RoboDK station: layout_PR2-2-7-bis.rdk

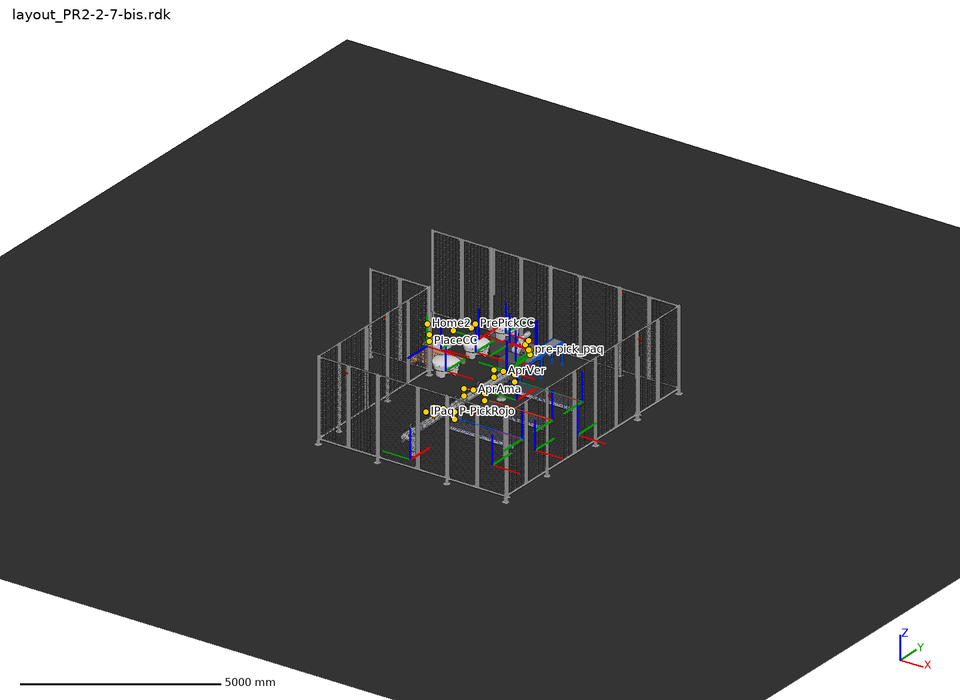
[picture v0: the station drawn from its stored meshes, robots at their saved joint values, targets as dots, program paths as lines]
Station def_pim_nigr (saved by RoboDK 5.9.4). Poses are relative to the parent item; angles as X-Y-Z fixed-axis rotations.
Station parameters (name, value as stored): IO_0, 1, IO_5, 1, IO_2, 1, IO_1, 1, IO_3, 0, 0, 0, 1, 0, 4, 0, SenyalSensor, 0, num_Pimiento, 0, num_Pimiento_Ama, 0, num_Pimiento_Rojo, 0, num_Pimiento_Verde, 0
  - folder Robots
    - frame D1Base at (200, 100, 1550) mm
      - robot D1 (model ABB IRB 360-1/1130 4D): 4 axes, payload 3 kg, reach 565 mm, repeatability 0.04 mm, weight 120 kg
          joint limits [-46.1, -46.1, -46.1, -36000] to [100.2, 100.2, 100.2, 36000]; home [0, 0, 0, 0]; saved at [70.365, 26.482, 30.889, 0]
        - tool GripR, TCP at (0, 0, 130) mm, size 75 x 83 x 136.1 mm
    - frame D2Base at (200, 1400, 1550) mm
      - robot D2 (model ABB IRB 360-1/1130 4D): 4 axes, payload 3 kg, reach 565 mm, repeatability 0.04 mm, weight 120 kg
          joint limits [-46.1, -46.1, -46.1, -36000] to [100.2, 100.2, 100.2, 36000]; home [0, 0, 0, 0]; saved at [70.365, 26.482, 30.889, 0]
        - tool GripA, TCP at (0, 0, 130) mm, size 75 x 83 x 136.1 mm
    - frame D3Base at (200, 2700, 1550) mm
      - robot D3 (model ABB IRB 360-1/1130 4D): 4 axes, payload 3 kg, reach 565 mm, repeatability 0.04 mm, weight 120 kg
          joint limits [-46.1, -46.1, -46.1, -36000] to [100.2, 100.2, 100.2, 36000]; home [0, 0, 0, 0]; saved at [70.365, 26.482, 30.889, 0]
        - tool GripV, TCP at (0, 0, 130) mm, size 75 x 83 x 136.1 mm
    - frame ABBPaq at (-570, 4240, -50) mm
      - robot ABBPaq (model ABB IRB 120-3/0.6): 6 axes, payload 3 kg, reach 580 mm, repeatability 0.01 mm, weight 25 kg
          modified DH rows (alpha deg, a mm, theta deg, d mm): 0, 0, 0, 290; -90, 0, -90, 0; 0, 270, 0, 0; -90, 70, 0, 302; 90, 0, 0, 0; -90, 0, 180, 72
          joint limits [-165, -110, -90, -160, -120, -400] to [165, 110, 70, 160, 120, 400]; home [0, 0, 0, 0, 0, 0]; saved at [84.8, 55.71, -70.13, 0, 104.39, 85]
        - tool ventosa_paq, TCP at (0, 0, 130) mm, size 75 x 83 x 136.1 mm
      - object Pedestal H24in (Type 1) at (-40, 0, -610) mm, size 400 x 400 x 609.6 mm, geometry from Pedestal-H24in-Type-1.sld
      - object SICK WL4S Laser Sensor at (638.65, -30.04, 245) mm, rotated rx 0 ry 0 rz 180 deg, size 683.3 x 45.2 x 12.5 mm, geometry from SICK-WL4S-Laser-Sensor.sld
    - frame ABBPallet at (-3120, 4660, -590) mm
      - robot ABBPallet (model ABB IRB 260): 4 axes, payload 30 kg, reach 1560 mm, repeatability 0.1 mm, weight 340 kg
          joint limits [-180, -28, -17, -300] to [180, 85, 119, 300]; home [0, 0, 0, 0]; saved at [-38.87, 11.87, -1.33, -35]
        - tool ventosa_pallet, TCP at (0, 30, 180) mm, size 239 x 147 x 184.9 mm
    - folder ProgCintas
      - program cintaROJO (3 instructions, listed below)
      - program cintaAMA (3 instructions, listed below)
      - program cintaVERDE (3 instructions, listed below)
  - folder Cintas
    - frame Conveyor Rojo at (2400, 300, 200) mm, rotated rx 0 ry 0 rz -180 deg
      - robot CRojo: 1 axes
          modified DH rows (alpha deg, a mm, theta deg, d mm): 0, 0, 0, 0 linear
          base shift (0, 0, 0) mm, rotated rx 0 ry 90 rz 0 deg
          joint limits [-500000] to [500000]; home [0]; saved at [0]
        - frame PRojo at (760, 220, -850) mm, rotated rx 0 ry 0 rz -180 deg
          - object PiRojo at (0, -5, 50) mm, rotated rx 180 ry 0 rz 180 deg, size 100 x 100 x 100 mm, geometry from Sphere-D100mm.sld
      - object SensorRojo at (1900, 0, 0) mm, rotated rx 0 ry 0 rz 90 deg, size 683.3 x 45.2 x 12.5 mm, geometry from SICK-WL4S-Laser-Sensor.sld
      - target IRojo (joint target) at (0, 0, 0) mm; joints [0] of CRojo
      - target FRojo (joint target) at (1900, 0, 0) mm; joints [1900] of CRojo
      - target P-PickRojo (Cartesian target) at (1900, 225, 300) mm, rotated rx 180 ry 0 rz 180 deg; joints [-31.271, 25.228, 30.105, 0] of D1
      - target PickRojo (Cartesian target) at (1900, 225, 100) mm, rotated rx 180 ry 0 rz 180 deg; joints [4.869, 47.636, 51.233, 0] of D1
      - target AprRojo (Cartesian target) at (2250, 225, 300) mm, rotated rx 180 ry 0 rz 180 deg; joints [4.316, -9.05, -2.968, 0] of D1
      - target P-PlaceRojo (Cartesian target) at (2532, 225, 250) mm, rotated rx 180 ry 0 rz 180 deg; joints [51.618, -4.676, 0.802, 0] of D1
      - target PlaceRojo (Cartesian target) at (2532, 225, 50) mm, rotated rx 180 ry 0 rz 180 deg; joints [70.365, 26.482, 30.889, 0] of D1
    - frame Conveyor Amarillo at (2400, 1600, 200) mm, rotated rx 0 ry 0 rz 180 deg
      - robot CAma: 1 axes
          modified DH rows (alpha deg, a mm, theta deg, d mm): 0, 0, 0, 0 linear
          base shift (0, 0, 0) mm, rotated rx 0 ry 90 rz 0 deg
          joint limits [-500000] to [500000]; home [0]; saved at [0]
        - frame PAma at (380, 220, -850) mm, rotated rx 0 ry 0 rz -180 deg
          - object PiAma at (0, 0, 50) mm, size 100 x 100 x 100 mm, geometry from Sphere-D100mm.sld
      - object SensorAma at (1900, 0, 0) mm, rotated rx 0 ry 0 rz 90 deg, size 683.3 x 45.2 x 12.5 mm, geometry from SICK-WL4S-Laser-Sensor.sld
      - target IAma (joint target) at (0, 0, 0) mm; joints [0] of CAma
      - target FAma (joint target) at (1900, 0, 0) mm; joints [1900] of CAma
      - target AprAma (Cartesian target) at (2250, 225, 300) mm, rotated rx 180 ry 0 rz 180 deg; joints [4.316, -9.05, -2.968, 0] of D2
      - target P-PickAma (Cartesian target) at (1900, 225, 300) mm, rotated rx 180 ry 0 rz 180 deg; joints [-31.271, 25.228, 30.105, 0] of D2
      - target PickAma (Cartesian target) at (1900, 225, 100) mm, rotated rx 180 ry 0 rz 180 deg; joints [4.869, 47.636, 51.233, 0] of D2
      - target P-PlaceAma (Cartesian target) at (2532, 225, 250) mm, rotated rx 180 ry 0 rz 180 deg; joints [51.618, -4.676, 0.802, 0] of D2
      - target PlaceAma (Cartesian target) at (2532, 225, 50) mm, rotated rx 180 ry 0 rz 180 deg; joints [70.365, 26.482, 30.889, 0] of D2
    - frame Conveyor Verde at (2400, 2900, 200) mm, rotated rx 0 ry 0 rz 180 deg
      - robot CVerde: 1 axes
          modified DH rows (alpha deg, a mm, theta deg, d mm): 0, 0, 0, 0 linear
          base shift (0, 0, 0) mm, rotated rx 0 ry 90 rz 0 deg
          joint limits [-500000] to [500000]; home [0]; saved at [0]
        - frame PVerd at (0, 220, -850) mm, rotated rx 0 ry 0 rz 180 deg
          - object PiVerd at (0, 0, 50) mm, size 100 x 100 x 100 mm, geometry from Sphere-D100mm.sld
      - object SensorVerde at (1900, 0, 0) mm, rotated rx 0 ry 0 rz 90 deg, size 683.3 x 45.2 x 12.5 mm, geometry from SICK-WL4S-Laser-Sensor.sld
      - target IVerde (joint target) at (0, 0, 0) mm; joints [0] of CVerde
      - target FVerde (joint target) at (1900, 0, 0) mm; joints [1900] of CVerde
      - target AprVer (Cartesian target) at (2250, 225, 300) mm, rotated rx 180 ry 0 rz 180 deg; joints [70.365, 26.482, 30.889, 0] of D3
      - target P-PickVer (Cartesian target) at (1900, 225, 300) mm, rotated rx 180 ry 0 rz 180 deg; joints [70.365, 26.482, 30.889, 0] of D3
      - target PickVer (Cartesian target) at (1900, 225, 100) mm, rotated rx 180 ry 0 rz 180 deg; joints [4.869, 47.636, 51.233, 0] of D3
      - target P-PlanceVer (Cartesian target) at (2532, 225, 250) mm, rotated rx 180 ry 0 rz 180 deg; joints [70.365, 26.482, 30.889, 0] of D3
      - target PlaceVerde (Cartesian target) at (2532, 225, 50) mm, rotated rx 180 ry 0 rz 180 deg; joints [70.365, 26.482, 30.889, 0] of D3
    - frame cinta_larga at (-40, -1070, -500) mm, rotated rx 0 ry 0 rz 89.89 deg
      - robot C1: 1 axes
          modified DH rows (alpha deg, a mm, theta deg, d mm): 0, 0, 0, 0 linear
          base shift (0, 0, 0) mm, rotated rx 0 ry 90 rz 0 deg
          joint limits [-900000] to [900000]; home [0]; saved at [0]
        - frame BasePIM at (4280, 95, 50) mm
    - frame Conveyor Paq at (-400, 4930, 0) mm, rotated rx 0 ry 0 rz -180 deg
      - robot CPaq: 1 axes
          modified DH rows (alpha deg, a mm, theta deg, d mm): 0, 0, 0, 0 linear
          base shift (0, 0, 0) mm, rotated rx 0 ry 90 rz 0 deg
          joint limits [-500000] to [500000]; home [0]; saved at [0]
        - frame CCBase at (800, 60, 0) mm
          - object CajaCerrada at (0, 0, 0) mm, size 252 x 305.4 x 216.7 mm, geometry from Box-12x10in-Closed.sld
        - frame FPaq at (0, 60, 0) mm
          - object CajaAbierta at (0, 0, 0) mm, size 274.3 x 328 x 215.5 mm, geometry from Box-12x10in-Open.sld
      - target IPaq (joint target) at (-18, 4855, 250) mm, rotated rx 180 ry 0 rz 180 deg; joints [70.365, 26.482, 30.889, 0] of D1
      - target FPaq (joint target) at (-18, 4855, 250) mm, rotated rx 180 ry 0 rz 180 deg; joints [70.365, 26.482, 30.889, 0] of D1
      - target pre-pick_paq (Cartesian target) at (-272, 690, 378) mm, rotated rx 180 ry 0 rz 0 deg; joints [0, 35.296, -44.946, 0, 99.65, 0] of ABBPaq
      - target pick_paq (Cartesian target) at (-272, 690, 258) mm, rotated rx 180 ry 0 rz 0 deg; joints [0, 29.358, -13.475, 0, 74.117, 0] of ABBPaq
      - target aprox_paq (Cartesian target) at (54.01, 442.2, 333.04) mm, rotated rx 180 ry 0.01 rz 34.1 deg; joints [34.1, 30.853, -29.576, 0, 88.712, 0] of ABBPaq
      - target pre-place_paq (Cartesian target) at (124.84, 193.82, 333.11) mm, rotated rx 179.97 ry 0 rz -0.2 deg; joints [84.8, 55.71, -70.13, 0, 104.39, 85] of ABBPaq
      - target place_paq (Cartesian target) at (124.84, 193.75, 68.06) mm, rotated rx 179.98 ry 0 rz -0.2 deg; joints [84.8, 53.502, -15.55, 0, 52.028, 85] of ABBPaq
  - folder P&P
    - program P&P_Rojo (26 instructions, listed below)
    - program P&P_Ama (26 instructions, listed below)
    - program P&P_Ver (26 instructions, listed below)
    - program P&P_Paq (20 instructions, listed below)
    - program Cajas (2 instructions, listed below)
  - folder Programas Python
    - Python program ACRojo (listed below)
    - Python program ACAma (listed below)
    - Python program ACVerde (listed below)
    - Python program ResetCinta (listed below)
    - Python program ACTodas (listed below)
    - Python program ACPaqPim (listed below)
    - Python program ResetPaq (listed below)
    - Python program ACCajaAbierta (listed below)
    - Python program ACCajaCerrada (listed below)
    - Python program P&P_CajaCerrada (listed below)
    - Python program MQTTListener (listed below)
    - Python program RobotController (listed below)
    - Python program STOP (listed below)
  - program Prog Princ (4 instructions, listed below)
  - Python program Reset total (listed below)
  - folder Objetos
    - frame PlaceCC at (-3250, 4210, -380) mm, rotated rx 90 ry 0 rz 0 deg
      - object Pallete at (0, 0, 0) mm, rotated rx 0 ry -90 rz -90 deg, size 800 x 1200 x 144.2 mm, geometry from Pallet-1200x800mm-Transverse.sld
    - frame PickCajaCerrada at (-1980, 4670, 0) mm, rotated rx 0 ry 0 rz 90 deg
      - target PrePickCC (Cartesian target) at (20, 125, 369) mm, rotated rx 180 ry 0 rz 90 deg; joints [0, 11.884, -1.332, 0] of ABBPallet
      - target PickCC (Cartesian target) at (50, 265, 209) mm, rotated rx 180 ry 0 rz 0 deg; joints [4.062, -0.234, 14.249, 94.062] of ABBPallet
      - target Home1 (Cartesian target) at (-616.94, 347.85, 369.01) mm, rotated rx 180 ry 0 rz 86.13 deg; joints [-38.87, 11.87, -1.33, -35] of ABBPallet
      - target Home2 (Cartesian target) at (-596.33, 1155.24, 331.73) mm, rotated rx 180 ry 0 rz 31.11 deg; joints [-93.89, -22.22, -1.33, -35] of ABBPallet
      - target PrePlaceCC (Cartesian target) at (-577.82, 1111.43, 41.13) mm, rotated rx 180 ry 0 rz 90 deg; joints [-87.263, -16.35, 27.423, -87.263] of ABBPallet
      - target PlaceCC (Cartesian target) at (-577.82, 1111.43, -158.87) mm, rotated rx 180 ry 0 rz 90 deg; joints [-87.263, -0.063, 54.303, -87.263] of ABBPallet
    - frame Conveyor Paq at (-30, 3530, -710) mm, rotated rx 0 ry 0 rz 90 deg
      - robot CRPaq: 1 axes
          modified DH rows (alpha deg, a mm, theta deg, d mm): 0, 0, 0, 0 linear
          base shift (0, 0, 0) mm, rotated rx 0 ry 90 rz 0 deg
          joint limits [-99999] to [9999999]; home [0]; saved at [0]
        - frame BasePaq at (-300, 100, 40) mm
          - object Paquete Pim at (0, 0, 0) mm, rotated rx 0 ry 90 rz 0 deg, size 81 x 81 x 243 mm, geometry from Cylinder-50x150mm.sld
    - object Maquina Plastificado at (-387, 3180, 0) mm, size 500 x 500 x 500 mm, geometry from Cube-500mm.sld
    - object Maquina Cerrado at (-1520, 4460, -190) mm, size 500 x 500 x 500 mm, geometry from Cube-500mm.sld
    - object CeldaDef at (-1000, -3500, -500) mm, size 7695.4 x 7756 x 2470 mm, geometry from CeldaDef.stl
    - object Floor at (0, 2530, -500) mm, rotated rx 0 ry 0 rz 90 deg, size 30000 x 30000 x 0 mm, geometry from Floor.sld
      - object Light (Red) at (-1230, 2420, 2250) mm, rotated rx -90 ry 0 rz 0 deg, size 75 x 75 x 139 mm, geometry from Light-Red.sld
        - object Light (Red) at (-3020, 0, -920) mm, rotated rx 0 ry -90 rz 0 deg, size 75 x 75 x 139 mm, geometry from Light-Red.sld
          - object Light (Red) at (-3900, 0, 0) mm, size 75 x 75 x 139 mm, geometry from Light-Red.sld
            - object Light (Red) at (-910, 0, -1820) mm, rotated rx -90 ry 0 rz 90 deg, size 75 x 75 x 139 mm, geometry from Light-Red.sld
              - object Light (Red) at (0, 3900, 0) mm, size 75 x 75 x 139 mm, geometry from Light-Red.sld
                - object Light (Red) at (0, 1820, -1810) mm, rotated rx -90 ry 0 rz 0 deg, size 75 x 75 x 139 mm, geometry from Light-Red.sld
                  - object Light (Red) at (0, 3900, 0) mm, size 75 x 75 x 139 mm, geometry from Light-Red.sld
    - frame PiEliminado at (-130, 3230, 210) mm
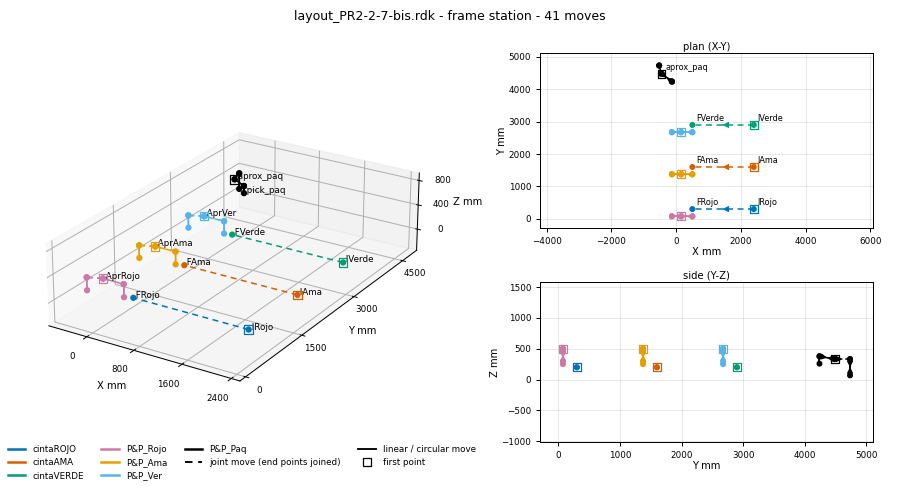
[picture p0: tool path of layout_PR2-2-7-bis.rdk in frame station, 41 of 41 moves have a stored position in this frame; points joined in program order, loops and branches not executed]

--- program cintaROJO (robot CRojo) ---
  Est. Ref.: Conveyor Rojo at (0, 0, 0) mm
  MoveJ (IRojo)
  MoveJ (FRojo)

--- program cintaAMA (robot CAma) ---
  Est. Ref.: Conveyor Amarillo
  MoveJ (IAma)
  MoveJ (FAma)

--- program cintaVERDE (robot CVerde) ---
  Est. Ref.: Conveyor Verde
  MoveJ (Inicio) -> target IVerde
  MoveJ (FinCinta) -> target FVerde

--- program P&P_Rojo (robot D1) ---
  Est. Ref.: Conveyor Rojo
  Est. herr: GripR
  Establecer velocidad (450.0 mm/s)
  MoveJ (aprox) -> target AprRojo
  MoveJ (pre-pick) -> target P-PickRojo
  Establecer velocidad (100.0 mm/s)
  Llamar ACRojo
  MoveL (pick) -> target PickRojo
  Pausa 3.5 s
  Set IO_0=1
  Wait IO_1=1
  Wait IO_2=1
  Adjuntar a GripR
  MoveL (pre-pick) -> target P-PickRojo
  Establecer velocidad (450.0 mm/s)
  MoveJ (aprox) -> target AprRojo
  MoveJ (pre-place) -> target P-PlaceRojo
  Establecer velocidad (100.0 mm/s)
  MoveL (place) -> target PlaceRojo
  Pausa 3.5 s
  Set IO_0=0
  Separar de GripR
  MoveL (pre-place) -> target P-PlaceRojo
  Establecer velocidad (450.0 mm/s)
  MoveJ (aprox) -> target AprRojo
  Reemplazar PRojo

--- program P&P_Ama (robot D2) ---
  Est. Ref.: Conveyor Amarillo
  Est. herr: GripA
  Establecer velocidad (450.0 mm/s)
  MoveJ (AprAma)
  MoveJ (PPickAma) -> target P-PickAma
  Establecer velocidad (100.0 mm/s)
  Llamar ACAma
  MoveL (PickAma)
  Pausa 3.5 s
  Set IO_1=1
  Wait IO_0=1
  Wait IO_2=1
  Adjuntar a GripA
  MoveL (P-PickAma)
  Establecer velocidad (450.0 mm/s)
  MoveJ (AprAma)
  MoveJ (P-PlaceAma)
  Establecer velocidad (100.0 mm/s)
  MoveL (PlaceAma)
  Pausa 3.5 s
  Set IO_1=0
  Separar de GripA
  MoveL (P-PlaceAma)
  Establecer velocidad (450.0 mm/s)
  MoveJ (AprAma)
  Reemplazar PAma

--- program P&P_Ver (robot D3) ---
  Est. Ref.: Conveyor Verde
  Est. herr: GripV
  Establecer velocidad (450.0 mm/s)
  MoveJ (AprVer)
  MoveJ (P-PickVer)
  Establecer velocidad (100.0 mm/s)
  Llamar ACVerde
  MoveL (PickVer)
  Pausa 3.5 s
  Set IO_2=1
  Wait IO_1=1
  Wait IO_0=1
  Adjuntar a GripV
  MoveL (P-PickVer)
  Establecer velocidad (450.0 mm/s)
  MoveJ (AprVer)
  MoveJ (P-PlanceVer)
  Establecer velocidad (100.0 mm/s)
  MoveL (PlaceVerde)
  Pausa 3.5 s
  Set IO_2=0
  Separar de GripV
  MoveL (P-PlanceVer)
  Establecer velocidad (450.0 mm/s)
  MoveJ (AprVer)
  Reemplazar PVerd

--- program P&P_Paq (robot ABBPaq) ---
  Est. Ref.: Conveyor Paq
  Est. herr: RobotiQ EPick Vacuum Gripper (1 Cup) -> ventosa_paq
  MoveJ (aprox_paq)
  MoveL (pre-pick_paq)
  Llamar ACPaqPim
  Establecer velocidad (850.0 mm/s)
  MoveL (pick_paq)
  Set IO_3=1
  Adjuntar a RobotiQ EPick Vacuum Gripper (1 Cup)
  MoveL (pre-pick_paq)
  Establecer velocidad (1000.0 mm/s)
  MoveJ (aprox_paq)
  MoveJ (pre-place_paq)
  Establecer velocidad (850.0 mm/s)
  MoveL (place_paq)
  Set IO_3=0
  Separar de ventosa_paq
  Reemplazar Paquete Pim
  MoveL (pre-place_paq)
  Llamar ResetPaq

--- program Cajas (robot ABBPaq) ---
  Llamar ACCajaAbierta
  Llamar ACCajaCerrada

--- Python program ACRojo ---
from robodk import robolink
from robodk import robomath

RDK = robolink.Robolink()

Cinta = RDK.Item('CRojo')
INCREMENTO_MM = 190
Pimiento = RDK.Item('PiRojo')
SistRefCinta = RDK.Item('PRojo')
Pimiento.setVisible(False)

if Cinta.Valid():
    Cinta.MoveJ(Cinta.Joints() + INCREMENTO_MM+190)

    Pimiento.Copy()
    PimientoCopia = RDK.Paste(SistRefCinta)
    PimientoCopia.setName('PiRojoB')
    PimientoCopia.setVisible(True)

    nPimiento = RDK.getParam('num_Pimiento_Rojo')
    if nPimiento is None:
        nPimiento = 0

    nPimiento += 1

    pose_pim_en_refcinta = (SistRefCinta.PoseAbs().inv() *Pimiento.PoseAbs())

    pose_final = (pose_pim_en_refcinta *robomath.transl((-INCREMENTO_MM * nPimiento)*2, 0, -850))

    PimientoCopia.setPose(pose_final)

    RDK.setParam('num_Pimiento_Rojo', nPimiento)

--- Python program ACAma ---
from robodk import robolink
from robodk import robomath

RDK = robolink.Robolink()

Cinta = RDK.Item('CAma')
INCREMENTO_MM = 190
Pimiento = RDK.Item('PiAma')
SistRefCinta = RDK.Item('PAma')
Pimiento.setVisible(False)
if Cinta.Valid():

    Cinta.MoveJ(Cinta.Joints() + INCREMENTO_MM+190)


    Pimiento.Copy()
    PimientoCopia = RDK.Paste(SistRefCinta)
    PimientoCopia.setName('PiRojoB')
    PimientoCopia.setVisible(True)
    # Leer contador
    nPimiento = RDK.getParam('num_Pimiento_Ama')
    if nPimiento is None:
        nPimiento = 0

    nPimiento += 1

    pose_pim_en_refcinta = (
        SistRefCinta.PoseAbs().inv() *
        Pimiento.PoseAbs()
    )

    pose_final = (pose_pim_en_refcinta *robomath.transl(INCREMENTO_MM * nPimiento*2, 0, 850))

    PimientoCopia.setPose(pose_final)

    RDK.setParam('num_Pimiento_Ama', nPimiento)

--- Python program ACVerde ---
from robodk import robolink
from robodk import robomath

RDK = robolink.Robolink()

Cinta = RDK.Item('CVerde')
INCREMENTO_MM = 190
Pimiento = RDK.Item('PiVerd')
SistRefCinta = RDK.Item('PVerd')
Pimiento.setVisible(False)
if Cinta.Valid():

    Cinta.MoveJ(Cinta.Joints() + INCREMENTO_MM+190)

    Pimiento.Copy()
    PimientoCopia = RDK.Paste(SistRefCinta)
    PimientoCopia.setName('PiRojoB')
    PimientoCopia.setVisible(True)
    nPimiento = RDK.getParam('num_Pimiento_Verde')
    if nPimiento is None:
        nPimiento = 0

    nPimiento += 1

    pose_pim_en_refcinta = (SistRefCinta.PoseAbs().inv() *Pimiento.PoseAbs())

    pose_final = (pose_pim_en_refcinta *robomath.transl(INCREMENTO_MM * nPimiento*2, 0, 850))

    PimientoCopia.setPose(pose_final)

    RDK.setParam('num_Pimiento_Verde', nPimiento)

--- Python program ResetCinta ---
from robodk import robolink

RDK = robolink.Robolink()

RDK.setParam('SenyalSensor', 0)
RDK.setParam('num_Pimiento_Rojo', 0)
RDK.setParam('num_Pimiento_Ama', 0)
RDK.setParam('num_Pimiento_Verde', 0)

items = RDK.ItemList(robolink.ITEM_TYPE_OBJECT)
for item in items:
    if item.Name().startswith('PiRojoB'):
        item.Delete()

cintas = ['CRojo', 'CAma', 'CVerde', 'C1','CPaq','CRPaq']

for nombre in cintas:
    cinta = RDK.Item(nombre)
    if cinta.Valid():
        cinta.setJoints([0])

--- Python program ACTodas ---
from robodk import robolink, robomath
import time

RDK = robolink.Robolink()

BasePim = RDK.Item('BasePim')

INCREMENTO_MM = 1200
TIEMPO_STEP = 0.5

# Lista de pimientos conocidos
pimientos = []
num_anterior = 0

while True:

    # -----------------------------
    # 1. Detectar pimientos actuales
    # -----------------------------
    actuales = []
    for obj in RDK.ItemList(robolink.ITEM_TYPE_OBJECT):
        try:
            if obj.Valid() and obj.Name().startswith('PiRojoB'):
                if obj.Parent() == BasePim:
                    actuales.append(obj)
        except:
            continue

    # Limpiar inválidos
    actuales = [p for p in actuales if p.Valid()]

    num_actual = len(actuales)

    # -----------------------------
    # 2. Detectar si hay NUEVOS
    # -----------------------------
    if num_actual > num_anterior:

        # Actualizar lista interna
        pimientos = actuales

        # Pose inversa
        try:
            base_pose_inv = BasePim.PoseAbs().inv()
        except:
            time.sleep(TIEMPO_STEP)
            continue

        # -----------------------------
        # 3. Mover TODOS una vez
        # -----------------------------
        for pim in pimientos:

            try:
                if not pim.Valid() or not pim.Visible():
                    continue
            except:
                continue

            try:
                pos_abs = pim.PoseAbs().Pos()
            except:
                continue

            # Movimiento en Y
            nueva_pose_abs = robomath.transl(
                pos_abs[0],
                pos_abs[1] + INCREMENTO_MM,
                pos_abs[2]
            )

            try:
                pim.setPoseAbs(nueva_pose_abs)
            except:
                continue

            # -----------------------------
            # 4. Comprobar límite en X
            # -----------------------------
            try:
                pose_rel = base_pose_inv * pim.PoseAbs()
                x_rel = pose_rel.Pos()[0]
            except:
                continue

            if x_rel > 0:
                try:
                    pim.setVisible(False)
                except:
                    continue

        # Actualizar contador
        num_anterior = num_actual

    # -----------------------------
    # Espera
    # -----------------------------
    time.sleep(TIEMPO_STEP+1)

--- Python program ACPaqPim ---
from robodk import robolink
from robodk import robomath

RDK = robolink.Robolink()

Cinta = RDK.Item('CRPaq')
SistRefCinta = RDK.Item('BasePaq')

INCREMENTO_MM = 880

if Cinta.Valid():

    joints = Cinta.Joints().list()
    joints[0] += INCREMENTO_MM

    Cinta.MoveJ(joints)

--- Python program ResetPaq ---
from robodk import robolink

RDK = robolink.Robolink()


cintas = ['CRPaq']

for nombre in cintas:
    cinta = RDK.Item(nombre)
    if cinta.Valid():
        cinta.setJoints([0])

--- Python program ACCajaAbierta ---
import time
from robodk import robolink, robomath

RDK = robolink.Robolink()

CajaBase = RDK.Item('CajaAbierta')
SistRefCinta = RDK.Item('FPaq')

DESPLAZAMIENTO_MM = 700
TIEMPO_TOTAL = 1.5
PASOS = 60

# Espera de 1.5 segundos ANTES de iniciar el ciclo
time.sleep(1.5)

if CajaBase.Valid() and SistRefCinta.Valid():

    # 1. Crear copia
    CajaBase.Copy()
    Caja = RDK.Paste(SistRefCinta)

    if not Caja.Valid():
        raise Exception("No se pudo crear la copia de la caja.")

    Caja.setName('Caja_Movil')

    pose_ini = Caja.Pose()

    # 2. Movimiento interpolado
    for i in range(PASOS):
        frac = (i + 1) / PASOS
        dx = DESPLAZAMIENTO_MM * frac

        nueva_pose = pose_ini * robomath.transl(dx, 0, 0)
        Caja.setPose(nueva_pose)

        time.sleep(TIEMPO_TOTAL / PASOS)

    # 3. Borrar la caja
    Caja.Delete()

--- Python program ACCajaCerrada ---
import time
from robodk import robolink
from robodk import robomath

RDK = robolink.Robolink()

CajaBase = RDK.Item('CajaCerrada')
SistRefCinta = RDK.Item('CCBase')

DESPLAZAMIENTO_MM = 910
TIEMPO_TOTAL = 1.5       # segundos
PASOS = 60               # más pasos = más fluido

if CajaBase.Valid() and SistRefCinta.Valid():

    # 1. Crear copia
    CajaBase.Copy()
    Caja = RDK.Paste(SistRefCinta)
    Caja.setName('Caja_Movil_2')

    pose_ini = Caja.Pose()

    # 2. Movimiento interpolado
    for i in range(PASOS):
        frac = (i + 1) / PASOS
        dx = DESPLAZAMIENTO_MM * frac

        pose = pose_ini * robomath.transl(dx, 0, 0)
        Caja.setPose(pose)

        time.sleep(TIEMPO_TOTAL / PASOS)

--- Python program P&P_CajaCerrada ---
# RoboDK API

# En este código se usa Divide y Vencerás, que es la parte de PRA pedida para la entreda de PR2, para calcular las posiciones de las cajas.

from robodk import robolink, robomath
import os

RDK = robolink.Robolink()

robot = RDK.Item('ABBPallet', robolink.ITEM_TYPE_ROBOT)

# Targets
target_Home1 = RDK.Item('Home1', robolink.ITEM_TYPE_TARGET)
target_Home2 = RDK.Item('Home2', robolink.ITEM_TYPE_TARGET)
target_PickCC = RDK.Item('PickCC', robolink.ITEM_TYPE_TARGET)
target_Pre_Pick = RDK.Item('PrePickCC', robolink.ITEM_TYPE_TARGET)
target_Pre_Place = RDK.Item('PrePlaceCC', robolink.ITEM_TYPE_TARGET)
target_PlaceCC = RDK.Item('PlaceCC', robolink.ITEM_TYPE_TARGET)

CajaCerrada = RDK.Item('Caja_Movil_2', robolink.ITEM_TYPE_OBJECT)
VentosaPallet = RDK.Item('ventosa_pallet', robolink.ITEM_TYPE_TOOL)

robot.setPoseTool(VentosaPallet)

# Variables
COLS = 4
FILAS = 3
DISTX = -310
DISTY = -260

TOTAL_POS = COLS * FILAS

FILE_INDEX = "paletizado_index.txt"


# Algoritmo Divide y Vencerás para generar posiciones


def dividir_pallet(x0, y0, cols, filas, distx, disty):

    # Caso base:
    # Si solo queda una posicion, devolverla
    if cols == 1 and filas == 1:
        return [(x0, y0)]

    posiciones = []

    # Divide horizontalmente si hay varias columnas
    if cols > 1:

        mitad = cols // 2

        # Subproblema izquierda
        posiciones += dividir_pallet(
            x0,
            y0,
            mitad,
            filas,
            distx,
            disty
        )

        # Subproblema derecha
        posiciones += dividir_pallet(
            x0 + mitad * distx,
            y0,
            cols - mitad,
            filas,
            distx,
            disty
        )

    # Divide verticalmente si solo queda una columna
    elif filas > 1:

        mitad = filas // 2

        # Subproblema superior
        posiciones += dividir_pallet(
            x0,
            y0,
            cols,
            mitad,
            distx,
            disty
        )

        # Subproblema inferior
        posiciones += dividir_pallet(
            x0,
            y0 + mitad * disty,
            cols,
            filas - mitad,
            distx,
            disty
        )

    return posiciones

# Generar todas las posiciones del pallet

posiciones_pallet = dividir_pallet(
    0,
    0,
    COLS,
    FILAS,
    DISTX,
    DISTY
)

# Leer indice de caja desde archivo

if os.path.exists(FILE_INDEX):

    with open(FILE_INDEX, "r") as f:
        index = int(f.read().strip())

else:
    index = 0


# Reiniciar pallet cuando se llena

if index >= TOTAL_POS:
    index = 0


# Obtener posicion actual

x_desplazamiento, y_desplazamiento = posiciones_pallet[index]


# Calcular poses de colocacion

base_pre = target_Pre_Place.Pose()
base_place = target_PlaceCC.Pose()

desplazamiento = robomath.transl(
    x_desplazamiento,
    y_desplazamiento,
    0
)

pose_pre = base_pre * desplazamiento
pose_place = base_place * desplazamiento


# Movimientos robot

robot.MoveJ(target_Home1)

robot.setSpeed(100, 100)
robot.MoveJ(target_Pre_Pick)

robot.setSpeed(25, 20)
robot.MoveL(target_PickCC)


# Coger caja

CajaCerrada.setParentStatic(RDK.ActiveStation())

VentosaPallet.AttachClosest('', 500)

robot.MoveL(target_Pre_Pick)


# Ir a pallet

robot.setSpeed(100, 100)

robot.MoveJ(target_Home2)
robot.MoveJ(pose_pre)

robot.setSpeed(25, 20)

robot.MoveL(pose_place)


# Soltar caja

robot.setDO(1, 0)

VentosaPallet.DetachAll()


# Salida segura

robot.MoveL(pose_pre)

robot.MoveJ(target_Home2)
robot.MoveJ(target_Home1)


# Guardar siguiente posicion

with open(FILE_INDEX, "w") as f:
    f.write(str(index + 1))

--- Python program MQTTListener ---
import paho.mqtt.client as mqtt
import RobotController as rc

# Configuracion MQTT
broker = "broker.hivemq.com"
port = 1883
user = "giirob"
passwd = "UPV2024"

# Sirve para los topics derivados de este
topic_commands = "pr2/sahuquillers/#"

# Cuando reciba mensaje
def on_message(mqttc, obj, msg):
    payload = msg.payload.decode("utf-8")
    topic = msg.topic
    rc.handle_message(mqttc, topic, payload)

# Conexion a MQTT
mqttc = mqtt.Client(mqtt.CallbackAPIVersion.VERSION2)
mqttc.on_message = on_message

mqttc.username_pw_set(username=user, password=passwd)
mqttc.connect(broker, port, 60)

mqttc.subscribe(topic_commands, 0)

mqttc.loop_forever()

--- Python program RobotController ---
from robodk import robolink
import time

# Conexión con RoboDK
RDK = robolink.Robolink()

# Contador de paquetes
contador_paq_robot = 0


def handle_message(mqttc, topic, payload):
    global contador_paq_robot

    payload = payload.strip().lower()

    # Cuando recibe en el topic "pr2/sahuquillers/paq" -> "paquete"
    if topic == "pr2/sahuquillers/paq" and payload == "paquete":

        contador_paq_robot += 1

        ejecutar_pp_paq()

        # Cada 6 paquetes ejecuta cajas
        if contador_paq_robot == 7:
            ejecutar_cajas()
            time.sleep(1) # para dejar que se vaya la caja
            ejecutar_pp_paq()
            contador_paq_robot = 0

    # Cuando recibe en el topic "pr2/sahuquillers/caja" -> "caja"
    elif topic == "pr2/sahuquillers/caja" and payload == "caja":
        print("-> Evento caja recibido")
        ejecutar_paletizado()

    # Cuando recibe en el topic "pr2/sahuquillers/stop" -> "stop"
    elif topic == "pr2/sahuquillers/stop" and payload == "stop":
        print("-> STOP recibido, ejecutando script STOP")
        ejecutar_stop()


# Programas de RoboDK

# pick and place de paquetes
def ejecutar_pp_paq():
    programa = RDK.Item("P&P_Paq", robolink.ITEM_TYPE_PROGRAM)

    if programa.Valid():
        if not programa.Busy():   # evita solapamientos
            programa.RunProgram()
    else:
        print("No se encontró el programa P&P_Paq en la estación.")

# paletizado de cajas
def ejecutar_paletizado():
    programa = RDK.Item("P&P_CajaCerrada")

    if programa.Valid():
        if not programa.Busy():
            programa.RunProgram()
    else:
        print("No se encontró el programa P&P_CajaCerrada en la estación.")

# cinta de cajas
def ejecutar_cajas():
    programa = RDK.Item("Cajas", robolink.ITEM_TYPE_PROGRAM)

    if programa.Valid():
        if not programa.Busy():
            programa.RunProgram()
    else:
        print("No se encontró el programa P&P_CajaCerrada en la estación.")

# parada de emergencia
def ejecutar_stop():
    programa = RDK.Item("STOP")

    if programa.Valid():
        programa.RunProgram()
    else:
        print("No se encontró el script STOP en la estación.")

--- Python program STOP ---
from robodk import robolink
# Para simular la parada de emergencia setea la vel de simulacion a 0
# Para continuar la simulación, setear a vel normal(5) a mano o con ResetTotal
RDK = robolink.Robolink()
RDK.setSimulationSpeed(0)

--- program Prog Princ (robot ABBPaq) ---
  Ejecutar P&P_Rojo
  Ejecutar P&P_Ama
  Ejecutar P&P_Ver
  Ejecutar ACTodas

--- Python program Reset total ---
from robodk import robolink

RDK = robolink.Robolink()
RDK.setSimulationSpeed(5)
programas = RDK.ItemList(robolink.ITEM_TYPE_PROGRAM)

for prog in programas:
    if prog.Busy():
        prog.Stop()

RDK.setParam('SenyalSensor', 0)
RDK.setParam('num_Pimiento_Rojo', 0)
RDK.setParam('num_Pimiento_Ama', 0)
RDK.setParam('num_Pimiento_Verde', 0)

items = RDK.ItemList(robolink.ITEM_TYPE_OBJECT)
for item in items:
    try:
        if item.Valid() and item.Name().startswith('PiRojoB'):
            item.Delete()
    except:
        continue

cintas = ['CRojo', 'CAma', 'CVerde', 'C1', 'CPaq', 'CRPaq']

for nombre in cintas:
    cinta = RDK.Item(nombre)
    if cinta.Valid():
        cinta.setJoints([0])

items = RDK.ItemList(robolink.ITEM_TYPE_OBJECT)
for item in items:
    if item.Name().startswith('Caja_Movil_2'):
        try:
            item.setJoints([0])
        except:
            item.Delete()
